PROGRAM Step_4_EvenEnder // Even Ender
VAR
	//-----------------Safety------------------
	LocalSafety_4 : BOOL;
	

END_VAR

// ---------- local safety ----------
LocalSafety_4 := EvenEnderMMP;

// ---------- defaults ----------

EvenEnderFWD := FALSE;


// ---------- Safety ----------
IF NOT Permissive OR NOT LocalSafety_4 THEN   // if anything unsafe, force the system to IDLE (state 0).
    Step4_State := 0;
END_IF



// -------------------------------Main sequence ---------------------------------
CASE Step4_State OF
// ---------------- IDLE/STOPPED ----------------
0: 
	
	EvenEnderFWD := FALSE;
	   
IF GradingVFD2FWD THEN         // Transition to RUN when the upstream grading conveyor (GradingVFD2) is running
	Step4_State := 10;
END_IF
	
	
	
// ----------------------- RUN ----------------------	
10:
	
	EvenEnderFWD := TRUE;     //EvenEnder motor to run forward.
	
IF NOT GradingVFD2FWD OR NOT Permissive OR NOT LocalSafety_4 THEN       // Return to IDLE if the upstream conveyor stops, or if a permissive/localsafety input is lost.
	EvenEnderFWD := FALSE;	
	Step4_State := 0;
		
END_IF
	
	
	
	
	
	
	
	
	
	
	
	
	
	
	
	
	
	
	
END_CASE

END_PROGRAM

(* stored: Version 1.1.0.1
   POU Step_4_EvenEnder: Id {0f8a0a75-c443-43fb-aa86-c1b5168b3cdf}, SpecialFunc None *)
